(* PLC project  *)

CONFIGURATION Empty_Module_10
END_CONFIGURATION
